FUNCTION Call_RFID

instRFIDInfeed(PermissionHardware := permissionHardware,
		   	   QuitError := instOperatingMode.StateOperatingMode.Quit.IsActive,
		   	   Reset := instOperatingMode.StateOperatingMode.Reset.IsActive,
		   	   SensorPartDetected := PartPresentConveyorInfeedEnd,
		   	   CommandID := RFIDFeedInReceivedCommandID,
		   	   ReadData := RFIDFeedInReadData,
		   	   Status := RFIDFeedInStatus,
		   	   ActorInstanceIndex := 0,
		   	   ActorInstanceName := 'FeedIn StackerCrane',
		   	   HMIInterface := HMI.hmiMachineSectionInterface,
		   	   FMReadingSerialNumber => finishedMessageReadSerialNumber,
		   	   ExecuteCommand => RFIDFeedInExecuteCommand,
		   	   Command => RFIDFeedInCommand,
		   	   WriteData => RFIDFeedInWriteData,
		   	   MemoryIndex => RFIDFeedInMemoryIndex);

reReadSerialNumber(CLK := PartPresentConveyorInfeedEnd AND NOT finishedMessageReadSerialNumber);			   
reFinishedMessageReadSerialNumber(CLK := finishedMessageReadSerialNumber);
instRFIDInfeed.ReadSerialNumber(reReadSerialNumber.Q);

IF reFinishedMessageReadSerialNumber.Q THEN
	readData.FeedInReadingPoint := RFIDFeedInReadData;
END_IF

END_FUNCTION

(* stored: Version 1.1.0.1
   POU Call_RFID: Id {d35ef5f1-c2a8-47ea-9556-60581a4cf8a1}, SpecialFunc None *)
